Staubli VAL3: readAll.pgx

public program readAll(num& x_nUserIn (dimensions=1), num& x_nValveOut (dimensions=1), num& x_nBasicIn (dimensions=1), num& x_nBasicOut (dimensions=1), num& x_nBasicIn2 (dimensions=1), num& x_nBasicOut2 (dimensions=1))
begin
  // Copyright (c) 2021, Institute for Factory Automation and Production Systems (FAPS)
  //
  // Licensed under the Apache License, Version 2.0 (the "License");
  // you may not use this file except in compliance with the License.
  // You may obtain a copy of the License at
  //
  //     http://www.apache.org/licenses/LICENSE-2.0
  //
  // Unless required by applicable law or agreed to in writing, software
  // distributed under the License is distributed on an "AS IS" BASIS,
  // WITHOUT WARRANTIES OR CONDITIONS OF ANY KIND, either express or implied.
  // See the License for the specific language governing permissions and
  // limitations under the License.


  x_nUserIn=dioGet(diUserIn)
  x_nValveOut=dioGet(diValveOut)

  if (bBasicIO1)
    x_nBasicIn=dioGet(diBasicIn)
    x_nBasicOut=dioGet(diBasicOut)
  else
    x_nBasicIn=0
    x_nBasicOut=0
  endIf

  if (bBasicIO2)
    x_nBasicIn2=dioGet(diBasicIn2)
    x_nBasicOut2=dioGet(diBasicOut2)
  else
    x_nBasicIn2=0
    x_nBasicOut2=0
  endIf

end
